INTERFACE I_Resettable

METHOD Reset : E_RpcMethodResponse
VAR_INPUT
    eRequester : E_Requester := E_Requester.PROG;
END_VAR
END_METHOD

END_INTERFACE

(* stored: Version 1.1.0.1, ProductVersion 3.1.4026.12
   Itf I_Resettable: Id {c0000002-0000-0000-0000-000000000001}
   Method Reset: Id {c0000002-0000-0000-1000-000000000001} *)
